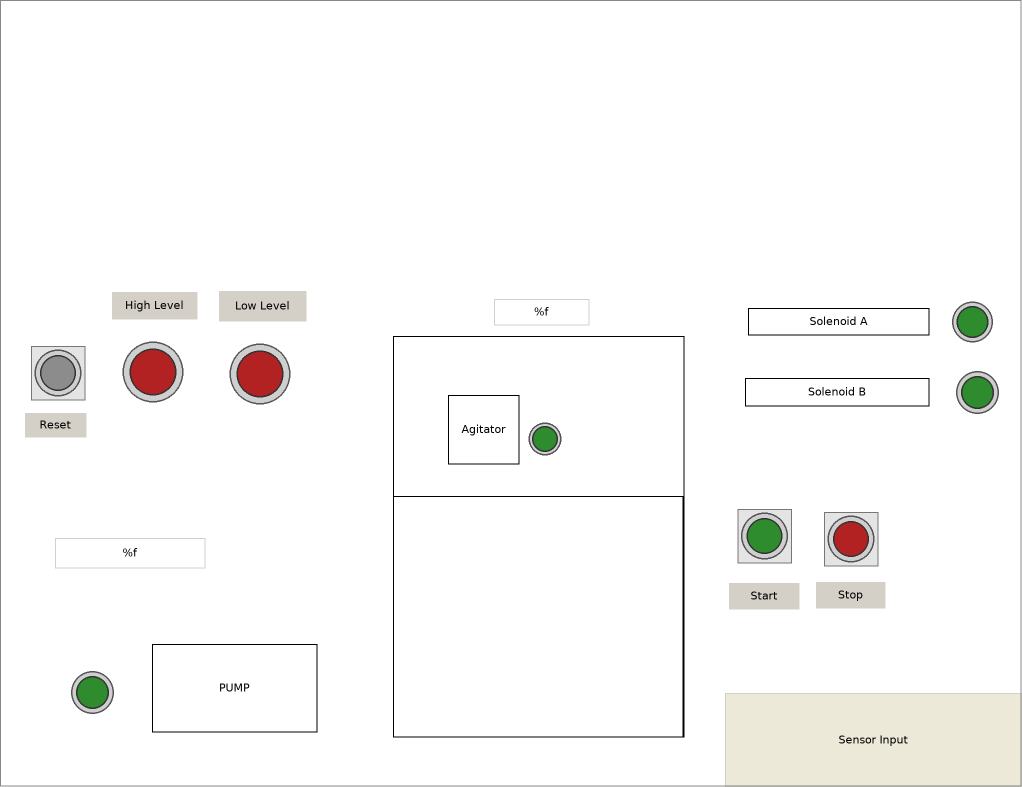
VISUALIZATION Visualization  // 1022x787
    Rectangle (393,336 291x401)
    Rectangle (393,496 290x241)
    Lamp1 (118,337 70x70), variable: Reservoir.bHighLevelAlarm, style: Lamp-Lamp1-Red
    Lamp1 (225,339 70x70), variable: Reservoir.bLowLevelAlarm, style: Lamp-Lamp1-Red
    Lamp1 (949,297 47x50), variable: Reservoir.bSolenoidALight, style: Lamp-Lamp1-Green
    Lamp1 (949,368 57x49), variable: Reservoir.bSolenoidBLight, style: Lamp-Lamp1-Green
    Lamp1 (526,413 38x52), variable: Reservoir.bAgitatorLight, style: Lamp-Lamp1-Green
    Lamp1 (68,665 49x55), variable: Reservoir.bPumpLight, style: Lamp-Lamp1-Green
    Rectangle (152,644 165x88), "PUMP"
    Rectangle (748,308 181x27), "Solenoid A"
    Rectangle (745,378 184x28), "Solenoid B"
    Rectangle (448,395 71x69), "Agitator"
    PushSwitch (31,345 54x56), variable: Reservoir.bResetButton, behaviour: TAP, style: Switch-PushSwitch-Gray
    PushSwitch (824,508 54x62), variable: Reservoir.bStopButton, behaviour: TAP, style: Switch-PushSwitch-Red
    PushSwitch (737,509 55x54), variable: Reservoir.bStartButton, behaviour: TAP, style: Switch-PushSwitch-Green
    Textfield (729,583 70x26), "Start"
    Textfield (816,582 69x26), "Stop"
    Textfield (25,413 61x24), "Reset"
    Textfield (112,292 85x27), "High Level"
    Textfield (219,291 87x30), "Low Level"
    Textfield (725,693 297x94), "Sensor Input", text variable: Reservoir.rSensorInput
        OnMouseDown: write the text variable via Default
    Textfield (55,538 150x30), "%f", text variable: Reservoir.rPumpOutput
    Textfield (494,299 95x26), "%f", text variable: Reservoir.rAgitatorOutput
END_VISUALIZATION

(* stored: Version 1.1.0.1, ProductVersion 3.1.4024.12
   Visu Visualization: Id {f0f33be0-7503-45b9-8b2f-92482d4d57a8} *)
